PROGRAM MAIN
VAR
	Counter : INT;
END_VAR

Counter := Counter + 1;

END_PROGRAM

(* stored: Version 1.1.0.1, ProductVersion 3.1.4024.6
   POU MAIN: Id {de4c17ca-6601-4dc2-9e9d-aef8e0f082a2}, SpecialFunc None *)
